{attribute 'qualified_only'}
VAR_GLOBAL
END_VAR

(* stored: Version 1.1.0.1
   GVL PartTracking_DB: Id {a31d5591-e7e2-43ca-b696-125a826acf42} *)
